// TwinCAT 3 PLC project Untitled1
// ProgramVersion: 3.1.4023.0
// libraries:
//   Tc2_MC2, * (Beckhoff Automation GmbH)
//   Tc2_MC2_Camming, * (Beckhoff Automation GmbH)
//   Tc2_MC2_Drive, * (Beckhoff Automation GmbH)
//   Tc2_Standard, * (Beckhoff Automation GmbH)
//   Tc2_System, * (Beckhoff Automation GmbH)
//   Tc3_Module, * (Beckhoff Automation GmbH)
//   Tc3_XTS_Utility, * (Beckhoff Automation GmbH)
// project tree:
//   GVLs/ GVL.TcGVL
//   / PlcTask.TcTTO
//   POUs/ MAIN.TcPOU

CONFIGURATION Untitled1
    RESOURCE PLC ON TwinCAT3
        TASK PlcTask(INTERVAL := T#10ms, PRIORITY := 20);
        PROGRAM MAIN WITH PlcTask : MAIN;
    END_RESOURCE
END_CONFIGURATION

// ---- GVLs/GVL.TcGVL
{attribute 'qualified_only'}
VAR_GLOBAL

	Movers : ARRAY[0..38] OF AXIS_REF;
	AsseNormale: AXIS_REF;

END_VAR

// ---- POUs/MAIN.TcPOU
PROGRAM MAIN
VAR CONSTANT
	nTub	: INT := 38;
	AlwaysTrue				: BOOL	:= TRUE;
	Alwaysfalse				: BOOL	:= FALSE;
END_VAR
VAR
	fbAxisActivete : ARRAY[0..nTub] OF MC_Power;
	fbAxisActivateNormale: MC_power;
	fbAxisStop		: ARRAY [0..ntub] OF MC_Stop;
	fbAxisStopNormale:	MC_Stop;
	McMoveAbsolute	: ARRAY[0..ntub] OF MC_MoveAbsolute;
	McMoveAbsoluteReal	: MC_moveAbsolute;
	McMoveVelocity		: ARRAY[0..ntub] OF MC_MoveVelocity;
	fbReset				: ARRAY[0..ntub] OF MC_Reset;
	
	i	: INT;
	j	: INT;
	bPower:BOOL;
	bAxisPower: BOOL;
	bAxisPowerNormale: BOOL;
	baxisActive: ARRAY[0..ntub] OF BOOL;
	bAxisNormalActive		: BOOL;
	bAxisStop: BOOL;
	bMoveAbsoluteEnable		: BOOL;
	bMoveAbsoluteEnableReale: BOOL;
	bMoveVelocityEnable		: BOOL;
	bMoveDone				: BOOL;
	bIsMoving				: BOOL;
	bInVelocity				: BOOL;
	bReset					: BOOL;
	bStop					: BOOL;
	bPLsStop				: BOOL;
	
	iMovePositionTub		: INT;
	iMovePositionNormale	: INT;
	iPosStop				: INT;
	
	rTrigStop				: R_TRIG;
	

END_VAR

//Read Status From Motion
FOR i := 0 TO nTub DO
	GVL.Movers[i].ReadStatus();
	GVL.AsseNormale.ReadStatus();
END_FOR

FOR i := 0 TO nTub DO
	fbReset[i](Axis:=GVl.Movers[i],
				Execute	:= bReset);
END_FOR

//Drive ON
FOR i := 0 TO nTub DO
		fbAxisActivete[i](Axis:=GVL.Movers[i],
						Enable:= bPower,
						Enable_Positive	:= AlwaysTrue,
						Enable_Negative	:= AlwaysTrue,
						Status=>baxisActive[i]);
END_FOR

//Normal Drive On
fbAxisActivateNormale(Axis:=GVL.AsseNormale,
							Enable:=bPower,
							Enable_Positive:= AlwaysTrue,
							Enable_Negative:= AlwaysTrue,
							Status=>bAxisNormalActive);
//Drives OFF	
FOR i := 0 TO nTub DO
	fbAxisStop[i](Axis:=GVL.Movers[i],
		Execute:= NOT bpower OR bStop);
END_FOR

IF fbAxisStop[0].Done THEN
	bStop		:= FALSE;
END_IF

//Asse Normale OFF
	fbAxisStopNormale(Axis:=GVL.AsseNormale,
		Execute:= NOT bpower);	
	
FOR i := 0 TO nTub DO	
	McMoveAbsolute[i](Axis:=	GVL.movers[i],
					execute:=bMoveAbsoluteEnable ,
					Position:= iMovePositionTub + (i*100),
					Velocity	:= 800 ,
					Acceleration	:= 80,
					Deceleration	:=80,
					Jerk			:= 100,
					Done=>bMoveDone,
					Active=>bIsMoving);
END_FOR

FOR i := 0 TO nTub DO	
	McMoveVelocity[i](Axis:=	GVL.movers[i],
					execute:=bMoveVelocityEnable ,
					Velocity	:= 800 ,
					Acceleration	:= 500,
					Deceleration	:=500,
					Jerk			:= 100,
					Direction		:= MC_Positive_Direction,
					InVelocity		=> bInVelocity,
					Active			=>bIsMoving);
END_FOR

IF bInVelocity THEN
	bMoveVelocityEnable	:= FALSE;
END_IF

 
McMoveAbsoluteReal(Axis:=	GVL.AsseNormale,
				execute:=bMoveAbsoluteEnableReale,
				Position:= iMovePositionNormale,
				Velocity	:= 80,
				Acceleration	:= 80,
				Deceleration	:=80,
				Jerk			:= 100,
				Done=>bMoveDone,
				Active=>bIsMoving);
				
				
(*				
//tentativo di fermarne uno al volo
IF (GVL.Movers[j].NcToPlc.ModuloActPos > iPosStop -100) AND (GVL.Movers[j].NcToPlc.ModuloActPos < iPosStop + 100) THEN
	bPLsStop	:= TRUE;
ELSE 
	bPLsStop	:= FALSE;
END_IF

rTrigStop(CLK:=bPLsStop,q=>);
IF rTrigStop.Q THEN
	fbAxisStop[j](Axis:=GVL.Movers[j],
		Execute:= TRUE,
		Deceleration:= 500);
	j:=j+1;
	j:=j MOD nTub;
END_IF
*)

END_PROGRAM
